// TIA Portal V18 export
TYPE "UDT_DLsDO"
// stored: IsFailsafeCompliant false
   STRUCT
      xDieselLineHeatingCmd : Array[1..2] of Bool;
      xDieselLinePumpEnable : Bool;
      xDieselLinePumpSelect : Bool;
      xDieselLineDayTankValve : Array[1..2] of Bool;
      Reserve : Array[1..2] of Bool;
   END_STRUCT;
END_TYPE
